FUNCTION_BLOCK FB_Sequenz_Testing
VAR_INPUT	
	Start			: BOOL 			:= FALSE;			// Start command
	Sequence_Name	: STRING(50) 	:= '';				// The name of the sequence
	Logging_active	: BOOL 			:= TRUE;			// The logging is default active. For deactivating set the variable to false.
END_VAR
VAR_OUTPUT
	Busy			: BOOL			:= FALSE;
	Finished		: BOOL			:= FALSE;			// The sequence is finished.
	Error			: BOOL			:= FALSE;			// Error during the sequence.
END_VAR
VAR_IN_OUT
	Step_list		: ARRAY [*] OF E_Test_step;	// Array with the sequence of steps
END_VAR
VAR
	Step_index		: DINT			:= 0;				// The current index of test step
	Step_state		: BYTE			:= 0;				// The internal state of the current test step
	Counter			: WORD			:= 0;				// Counter variable for internal use
	
	Name			: STRING(50)	:= '';				// The current sequence name. The name is saved once by start of the sequence.
	
	Data			: ARRAY [0..255] OF BYTE;
	CAN_Object		: ST_CAN_Object;	
	SDO_READ		: FB_SDO_READ;
	SDO_WRITE		: FB_SDO_WRITE;
	Write_busy		: BOOL 			:= FALSE;			// A writing process is running. After finishing the process the next test step is started
	Write_sequence	: BOOL			:= FALSE;			// If this Flag is set, the internal step state is increased. Otherwise the test step is finished after the write process.
	
	Next_Step_state	: BOOL 			:= FALSE;			// Increase the internal state of the test step
	Step_Finished	: BOOL 			:= FALSE;			// Switch to the next test step
	Error_step		: DINT 			:= -1;				// List index of the test state, at which an error is occured
	
	Current_Statemachine_state: E_Statemachine_State;	// The current State machine state
	
	Timeout_Counter	: INT			:= 0;				// Timeout Counter
	Timeout_Max		: INT			:= 0;				// Value at which the timeout counter is triggered (x 10 ms)

	Wait_Counter	: INT			:= 0;				// Wait Counter
	Wait_Step_Finish: BOOL			:= TRUE;			// True: The step is finished after the waiting time. False: The status counter in the step is increased after the waiting time.
	Wait_Time		: INT			:= 0;				// Value at which the wait counter is triggered (x 10 ms)

	Message			: STRING(60)	:= '';				// This message is send at the end of the FB
END_VAR

// Start / Reset
IF Start AND NOT Busy THEN
	Step_index		:= 0;
	Step_state 		:= 0;	
	Finished		:= FALSE;
	Error			:= FALSE;
	Error_step		:= -1;
 	Busy 			:= TRUE;	
	Name 			:= Sequence_Name;
	IF Sequence_Name = '' AND Logging_active THEN
		GLB.Logger(Message:='Start sequence');
	ELSE
		GLB.Logger(Message:=CONCAT('Start sequence: ', Sequence_Name)); 
	END_IF
END_IF


IF Busy THEN
	// Reached end?
	IF (Step_index > UPPER_BOUND(Step_list, 1)) OR (Error_step > -1) THEN
		Busy 		:= FALSE;
		Finished 	:= TRUE;
		IF Error_step = -1 AND Logging_active THEN
			GLB.Logger(Message:='Sequence successful', SaveFlag:=TRUE);
			Error	:= FALSE;
		ELSE	
			GLB.Logger(Message:='Sequence failed', SaveFlag:=TRUE);			
			Error	:= TRUE;		
		END_IF
				
	ELSE
		// Get the current state of the State machine
		Current_Statemachine_state 			:= GET_STATE(PDO.Statusword);
			
		// Processing the individual test steps  
		CASE Step_list[Step_index] OF
		
			// **** Change of state machine state *****
			// Switch directly to state 'Switch on disabled' -> Set Controlword to 0
			E_Test_step.Switch_on_disabled:
				CASE Step_state OF
					0:	// Set Controlword to 0
						PDO.Controlword			:= E_Statemachine_Transition_Controlword.Switch_on_disabled;
						Message					:= 'Switch to state Switch on disabled';		
						Next_Step_state			:= TRUE;
					
					1:	// Wait until state 'Switch on disabled'
						IF Current_Statemachine_state = E_Statemachine_State.Switch_on_disabled THEN		Step_Finished := TRUE;	END_IF	
				END_CASE	
				
			// Switch directly to state 'Quick stop active' -> Set Controlword to 2		
			E_Test_step.Quick_stop_active:
				CASE Step_state OF
					0:	// Set Controlword to 2
						PDO.Controlword			:= E_Statemachine_Transition_Controlword.Quick_stop_active;
						Message					:= 'Switch to state Quick stop active';		
						Next_Step_state			:= TRUE;
					
					1:	// Wait until state 'Quick stop active'
						IF Current_Statemachine_state = E_Statemachine_State.Quick_stop_active THEN			Step_Finished := TRUE;	END_IF
				END_CASE
													
			// Switch directly to state 'Ready to switch on' -> Set Controlword to 6		
			E_Test_step.Ready_to_switch_on:
				CASE Step_state OF
					0:	// Set Controlword to 6
						PDO.Controlword			:= E_Statemachine_Transition_Controlword.Ready_to_switch_on;
						Message					:= 'Switch to state Ready to switch on';			
						Next_Step_state			:= TRUE;				
				
					1:	// Wait until state 'Ready to switch on'
						IF Current_Statemachine_state = E_Statemachine_State.Ready_to_switch_on THEN		Step_Finished := TRUE;	END_IF
				END_CASE
													
			// Switch directly to state 'Switched on' -> Set Controlword to 7			
			E_Test_step.Switched_on:				
				CASE Step_state OF
					0:	// Set Controlword to 7
						PDO.Controlword			:= E_Statemachine_Transition_Controlword.Switched_on;
						Message					:= 'Switch to state Switched on';				
						Next_Step_state			:= TRUE;
					
					1:	// Wait until state 'Switched on'
						IF Current_Statemachine_state = E_Statemachine_State.Switched_on THEN				Step_Finished := TRUE;	END_IF
				END_CASE
													
			// Switch directly to state 'Operation enabled' -> Set Controlword to F		
			E_Test_step.Operation_enabled:				
				CASE Step_state OF
					0:	// Set Controlword to F
						PDO.Controlword			:= E_Statemachine_Transition_Controlword.Operation_enabled;
						Message					:= 'Switch to state Operation enabled';			
						Next_Step_state			:= TRUE;
					
					1:	// Wait until state 'Operation enabled'
						IF Current_Statemachine_state = E_Statemachine_State.Operation_enabled THEN			Step_Finished := TRUE;	END_IF
				END_CASE													
			// ****************************************	
						
			// ***** Change of Mode of Operation ******
			// Set Mode of Operation to 'No mode'
			E_Test_step.No_Mode:
				CASE Step_state OF
					0:
						PDO.Mode_of_operation	:= E_Mode_of_Operation.No_mode_active;
						Message					:= 'Set Mode of Operation to "No mode"';		
						Next_Step_state			:= TRUE;
					
					1:	// Wait until mode 'No mode'
						IF PDO.Mode_of_operation_display = E_Mode_of_Operation.No_mode_active THEN			Step_Finished := TRUE;	END_IF				
				END_CASE
						
			// Set Mode of Operation to 'Profile Position Mode'
			E_Test_step.Mode_PPM:
				CASE Step_state OF
					0:	
						PDO.Mode_of_operation	:= E_Mode_of_Operation.Profile_position_mode;
						Message					:= 'Set Mode of Operation to "Profile Position Mode"';			
						Next_Step_state			:= TRUE;
					
					1:	// Wait until mode 'Profile Position Mode'
						IF PDO.Mode_of_operation_display = E_Mode_of_Operation.Profile_position_mode THEN	Step_Finished := TRUE;	END_IF				
				END_CASE
								
			// Set Mode of Operation to 'Velocity Mode'
			E_Test_step.Mode_VM:
				CASE Step_state OF
					0:
						PDO.Mode_of_operation	:= E_Mode_of_Operation.Velocity_mode;
						Message					:= 'Set Mode of Operation to "Velocity Mode"';			
						Next_Step_state			:= TRUE;
					
					1:	// Wait until mode 'Velocity Mode'
						IF PDO.Mode_of_operation_display = E_Mode_of_Operation.Velocity_mode THEN			Step_Finished := TRUE;	END_IF		
				END_CASE
			
			// Set Mode of Operation to 'Profile Velocity Mode'
			E_Test_step.Mode_PVM:
				CASE Step_state OF
					0:
						PDO.Mode_of_operation	:= E_Mode_of_Operation.Profile_velocity_mode;
						Message					:= 'Set Mode of Operation to "Profile Velocity Mode"';			
						Next_Step_state			:= TRUE;
					
					1:	// Wait until mode 'Profile Velocity Mode'
						IF PDO.Mode_of_operation_display = E_Mode_of_Operation.Profile_velocity_mode THEN	Step_Finished := TRUE;	END_IF		
				END_CASE
										
			// Set Mode of Operation to 'Profile Torque Mode'
			E_Test_step.Mode_PTM:
				CASE Step_state OF
					0:
						PDO.Mode_of_operation	:= E_Mode_of_Operation.Profile_torque_mode;
						Message					:= 'Set Mode of Operation to "Profile Torque Mode"';		
						Next_Step_state			:= TRUE;
					
					1:	// Wait until mode 'Profile Torque Mode'
						IF PDO.Mode_of_operation_display = E_Mode_of_Operation.Profile_torque_mode THEN		Step_Finished := TRUE;	END_IF		
				END_CASE
				
			// Set Mode of Operation to 'Homing Mode'
			E_Test_step.Mode_HM:
				CASE Step_state OF
					0:
						PDO.Mode_of_operation	:= E_Mode_of_Operation.Homing_mode;
						Message					:= 'Set Mode of Operation to "Homing mode"';
						Next_Step_state			:= TRUE;
					
					1:	// Wait until mode 'Homing Mode'
						IF PDO.Mode_of_operation_display = E_Mode_of_Operation.Homing_mode THEN				Step_Finished := TRUE;	END_IF		
				END_CASE
										
			// Set Mode of Operation to 'Interpolated Position Mode'
			E_Test_step.Mode_IPM:
				CASE Step_state OF
					0:
						PDO.Mode_of_operation	:= E_Mode_of_Operation.Interpolated_position_mode;
						Message					:= 'Set Mode of Operation to "Interpolated Position Mode"';
						Next_Step_state			:= TRUE;
					
					1:	// Wait until mode 'Interpolated Position Mode'
						IF PDO.Mode_of_operation_display = E_Mode_of_Operation.Interpolated_position_mode THEN	Step_Finished := TRUE;	END_IF		
				END_CASE
			// ****************************************	
						
			// ************** Init steps **************	
			// Set the factor group to use rpm as user-defined velocity unit
			E_Test_step.Factor_group_rpm:
				Write_busy := TRUE;
				CASE Step_state OF
					0:	// Set ...
						Write_sequence := TRUE;
						DWORD_TO_BYTE_ARRAY(4096, Data);			
						CAN_Object 		:= DS402_Object_List.Velocity_Factor_Numerator;
						
					2:	// Set ...
						Write_sequence := FALSE;					
						DWORD_TO_BYTE_ARRAY(60, Data);			
						CAN_Object 		:= DS402_Object_List.Velocity_Factor_Divisor;
						
						
						
				END_CASE	
			// ****************************************	
			
			// ************ Setting values ************	
			// Set 'Velocity_window' to value 30
			E_Test_step.Velocity_window_30rpm:
				CASE Step_state OF
					0:
						DWORD_TO_BYTE_ARRAY(30, Data);			
						CAN_Object 		:= DS402_Object_List.Velocity_window;
						Message 		:= 'Set Velocity_window to 30';					
						Write_busy		:= TRUE;		
				END_CASE
			
			// Set 'Velocity window time' to value 100
			E_Test_step.Velocity_window_100ms:
				CASE Step_state OF
					0:
						DWORD_TO_BYTE_ARRAY(100, Data);			
						CAN_Object 		:= DS402_Object_List.Velocity_window_time;
						Message			:= 'Set Velocity window time to 100';					
						Write_busy		:= TRUE;
				END_CASE
				
			// Set 'Profile acceleration' to value 1000
			E_Test_step.Acceleration_1000:
				CASE Step_state OF
					0:
						DWORD_TO_BYTE_ARRAY(1000, Data);			
						CAN_Object 		:= DS402_Object_List.Profile_acceleration;
						Message			:= 'Set Profile acceleration to 1000';
						Write_busy		:= TRUE;	
				END_CASE
				
			// Set 'Profile deceleration' to value 1000			
			E_Test_step.Deceleration_1000:
				CASE Step_state OF
					0:
						DWORD_TO_BYTE_ARRAY(1000, Data);	
						CAN_Object 		:= DS402_Object_List.Profile_deceleration; 				
						Message			:= 'Set Profile deceleration to 1000';
						Write_busy		:= TRUE;
				END_CASE
				
			// Set 'Profile velocity' to value 1000			
			E_Test_step.PPM_Velocity_1000:
				CASE Step_state OF
					0:
						DWORD_TO_BYTE_ARRAY(1000, Data);			
						CAN_Object 		:= DS402_Object_List.Profile_velocity;
						Message			:= 'Set Profile velocity to 1000';					
						Write_busy		:= TRUE;	
				END_CASE
	
			// Set 'Target velocity' to value 1000
			E_Test_step.PVM_Velocity_1000:
				CASE Step_state OF
					0:	
						DWORD_TO_BYTE_ARRAY(1000, Data);			
						CAN_Object 		:= DS402_Object_List.Target_velocity;
						Message			:= 'Set Target velocity to 1000';
						Write_busy		:= TRUE;
				END_CASE		
			// ****************************************	
							
			// *********** Check conditions ***********
			// Check if the 'Target reached' bit in statusword is set within 200 ms
			E_Test_step.Check_Statusword_Target_reached_200ms:
				Timeout_Max 		:= 20;
				IF (PDO.Statusword AND E_Statusword_Bits.Target_reached) = E_Statusword_Bits.Target_reached THEN
					Message			:= 'Target reached bit is set';
					Step_Finished	:= TRUE;					
				END_IF	
			// ****************************************				
			
			// ************ Waiting times *************
			E_Test_step.Wait_10ms:		IF Step_state = 0 THEN	Wait_Time := 1; 	Message := 'Wait Time 10 ms is running';	Next_Step_State:=TRUE; END_IF
			E_Test_step.Wait_50ms:		IF Step_state = 0 THEN	Wait_Time := 5; 	Message := 'Wait Time 50 ms is running';	Next_Step_State:=TRUE; END_IF
			E_Test_step.Wait_100ms:		IF Step_state = 0 THEN	Wait_Time := 10; 	Message := 'Wait Time 100 ms is running';	Next_Step_State:=TRUE; END_IF
			E_Test_step.Wait_250ms:		IF Step_state = 0 THEN	Wait_Time := 25; 	Message := 'Wait Time 250 ms is running';	Next_Step_State:=TRUE; END_IF
			E_Test_step.Wait_500ms:		IF Step_state = 0 THEN	Wait_Time := 50; 	Message := 'Wait Time 500 ms is running';	Next_Step_State:=TRUE; END_IF
			E_Test_step.Wait_1000ms:	IF Step_state = 0 THEN	Wait_Time := 100; 	Message := 'Wait Time 1 s is running';		Next_Step_State:=TRUE; END_IF
			E_Test_step.Wait_2500ms:	IF Step_state = 0 THEN	Wait_Time := 250; 	Message := 'Wait Time 2.5 s is running';	Next_Step_State:=TRUE; END_IF
			// Feel free to create your own needed wait times :-)
			// ****************************************		
						
			ELSE
				// unknown steps -> next step
				Message				:= CONCAT(CONCAT('FB_Start_Testing: ERROR, unknown test step (', DINT_TO_STRING(Step_index)), ')');
				Step_Finished		:= TRUE;
	
		END_CASE
		
		// Waiting time. Active, if Wait_Time is greater than 0
		IF Wait_Time > 0 THEN
			Wait_Counter			:= Wait_Counter + 1;	
			IF Wait_Counter >= Wait_Time THEN
				Message				:= 'Waiting time expired';			
				IF Wait_Step_Finish THEN 
					Step_Finished	:= TRUE;
				ELSE
					Next_Step_state	:= TRUE;
				END_IF
			END_IF
		END_IF
		
		// SDO Write process is running. This generell function is used, if Write_busy is set.
		IF Write_busy THEN
			IF Step_state.0 = 0 THEN
				// Start writing
				SDO_Write(
					ADSNetID		:= GLB.ADSNetID_CAN,				
					PortNr 		 	:= 16#1000 + GLB.NodeID,
					CO_Index 		:= CAN_Object.Index,
					CO_SubIndex 	:= CAN_Object.Subindex,
					DataLength 		:= CAN_Object.Length,
					WriteData		:= Data,
					StartWriting	:= TRUE	);
				Next_Step_state	:= TRUE;								
			ELSE
				// Wait for finishing
				SDO_Write(StartWriting:=FALSE);
				IF SDO_WRITE.WriteDataFinished THEN
					Write_busy			:= FALSE;
					IF SDO_WRITE.Error = 0 THEN									
						IF Write_sequence THEN
							Next_step_state	:= TRUE;
						ELSE						
							Step_Finished	:= TRUE;
						END_IF;
					ELSE
						Message			:= CONCAT('ERROR: Write failed, Errornumber: ', DWORD_TO_HEXSTR(SDO_WRITE.Error, 8, FALSE));
						Error_step		:= Step_index;		
					END_IF	
					SDO_Write();	
				END_IF
			END_IF
		END_IF
		
		// Next Test step
		IF Step_Finished THEN
			IF Message = '' THEN Message := 'OK'; END_IF
			Step_Finished 			:= FALSE;
			Step_index				:= Step_index + 1;
			Step_state 				:= 0;
			Wait_Counter			:= 0;
			Wait_Time				:= 0;
			Wait_Step_Finish		:= TRUE;
			Write_sequence			:= FALSE;
			Timeout_Counter			:= 0;
			Timeout_Max 			:= 10;			// Set Timeout to a default value of 10 (= 100 ms)
			
		// Next internal state of the test step			
		ELSIF Next_Step_state THEN
			Next_Step_state			:= FALSE;
			Step_state				:= Step_state + 1;
			Timeout_Counter			:= 0;	
		
		// Timeout
		ELSE
			IF Timeout_Max > 0 THEN
				IF Timeout_Counter >= Timeout_Max THEN
					Message			:= CONCAT(CONCAT('Timeout triggered (', INT_TO_STRING(Timeout_Max * 10)), ' ms)');
					Error_step		:= Step_index;
				END_IF
				Timeout_Counter	:= Timeout_Counter + 1;	
			END_IF
		END_IF
	END_IF
	
	
	// Log message
	IF Message <> '' AND Logging_active  THEN
		GLB.Logger(Message:=Message);
		Message := '';
	END_IF
END_IF

END_FUNCTION_BLOCK

(* stored: Version 1.1.0.1, ProductVersion 3.1.4024.11
   POU FB_Sequenz_Testing: Id {54508373-3272-4d80-8bd4-d80740e4ba69}, SpecialFunc None *)
